// TIA Portal project "TestCase2_S1200_Met_Fouten" (V18)

(* hardware
DEVICE "S7-1200 station_1"  S7-1200 Station
   slot 0: "Rack_0"  S7-1200 Rack  Rack  V1.0
   slot 1: "PLC_1"  CPU 1212C DC/DC/DC  6ES7 212-1AE40-0XB0  V4.6
*)

// ===== PLC "PLC_1"  CPU 1212C DC/DC/DC =====

VAR_GLOBAL   // PLC tag table "Default tag table"
   "A" AT %I0.0 : Bool;
   "X" AT %Q0.0 : Bool;
   "Y" AT %Q0.1 : Bool;
END_VAR

DATA_BLOCK "Data_block_1_Inputs"   // DB1
{ S7_Optimized_Access := 'FALSE' }
VERSION : 0.1
   VAR
      "A" : Bool;
   END_VAR
BEGIN
END_DATA_BLOCK

DATA_BLOCK "Data_block_2_Outputs"   // DB2
{ S7_Optimized_Access := 'FALSE' }
VERSION : 0.1
   VAR
      X : Bool;
      Y : Bool;
   END_VAR
BEGIN
END_DATA_BLOCK

// folder: System blocks/Program resources

DATA_BLOCK "IEC_Timer_0_DB"   // DB3
{ S7_Optimized_Access := 'TRUE' }
AUTHOR : Simatic
FAMILY : IEC
NAME : IEC_TMR
VERSION : 1.0
// stored: InstanceOfName IEC_TIMER
"IEC_TIMER"
BEGIN
END_DATA_BLOCK

DATA_BLOCK "IEC_Timer_0_DB_1"   // DB4
{ S7_Optimized_Access := 'TRUE' }
AUTHOR : Simatic
FAMILY : IEC
NAME : IEC_TMR
VERSION : 1.0
// stored: InstanceOfName IEC_TIMER
"IEC_TIMER"
BEGIN
END_DATA_BLOCK

// folder: (top level)

ORGANIZATION_BLOCK "Main"   // OB1, FBD, ProgramCycle
TITLE = "Main Program Sweep (Cycle)"
{ S7_Optimized_Access := 'TRUE' }
VERSION : 0.1
   VAR_INPUT
      Initial_Call : Bool;   // Initial call of this OB
      Remanence : Bool;   // =True, if remanent data are available
   END_VAR
BEGIN

REGION Network 1
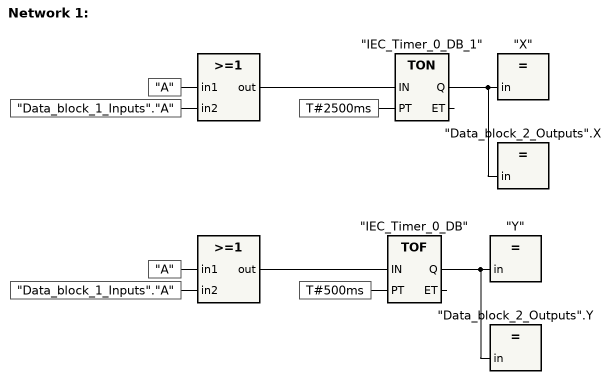
   "IEC_Timer_0_DB_1".TON(IN := "A" OR "Data_block_1_Inputs"."A", PT := T#2500ms);
   "X" := "IEC_Timer_0_DB_1".Q;
   "Data_block_2_Outputs".X := "IEC_Timer_0_DB_1".Q;
   "IEC_Timer_0_DB".TOF(IN := "A" OR "Data_block_1_Inputs"."A", PT := T#500ms);
   "Y" := "IEC_Timer_0_DB".Q;
   "Data_block_2_Outputs".Y := "IEC_Timer_0_DB".Q;
END_REGION
END_ORGANIZATION_BLOCK